{region '#Template'}
	{attribute 'Category' := 'DUTs'}
	{attribute 'Version' := '0.0.1.0'}
	{attribute 'Tags' := 'Plant, AC, OpMod'}
	{attribute 'Description' := 'Betriebsart Klimaanlage // Operation Mode Air Conditioning'}
{endregion}
{attribute qualified_only}
TYPE E_BA_AC_OpMod02 :
(
    Invalid							:= 0,
    eOff							:= 1,	// Aus//Off
    eStep1							:= 2,	// Stufe 1						// Step 1
    eStep2							:= 3,	// Stufe 2						// Step 2
    eStep3							:= 4,	// Stufe 3						// Step 3
    eEmergency						:= 5,	// Notfall						// Emergency
    eFrost							:= 6,	// Frost						// Frost
    eSmokeExtractionProgramm		:= 7,	// Entrauchung Programm			// Smoke extraction program
    eSmokeExtractionSupplyAir		:= 8,	// Entrauchung Zuluft			// Smoke extraction supply air
    eSmokeExtractionExhaustAir		:= 9,	// Entrauchung Fortluft			// Smoke extraction exhaust air
    eFire							:= 10,	// Feuer						// Fire
    eNightCooling					:= 11,	// Nachtkühlung					// Night cooling
    eCoolDownProtection				:= 12,	// Stützbetrieb,Auskühlschutz	// Cool down protection
    eOverHeatingProtection			:= 13,	// Überhitzungsschutz			// Over heating protection
    eAlarm							:= 14,	// Störung						// Alarm
    eForcedVentilation				:= 15,	// Zwangsbelüftung				// Forced ventilation
    eCentralSwitchOff				:= 16	// Zentralabschaltung			// Central switch-off
) UDINT;
END_TYPE

(* stored: Version 1.1.0.1, ProductVersion 3.1.4024.6
   DUT E_BA_AC_OpMod02: Id {85bf0050-54d4-47be-9674-976942f742d4} *)
